FUNCTION_BLOCK FB_Conveyor
VAR CONSTANT
	sCycleStateTextDef: ARRAY[0..10]  OF STRING :=	
		['State 0: Wait for Start',
		'State 1: Start conveyor',
		'State 2: Start Gantries',
		'State 3: Spare',
		'State 4: Spare',
		'State 5: Spare',
		'State 6: Belt running, control speed','7','8','9',
		'State 10: Error'];
	
	tCycleStateTimeouts: ARRAY[0..10] OF TIME := 
		[T#10S,T#10S,T#60S,T#10S,T#10S,T#10S,T#10S,T#10S,T#10S,T#10S,
		T#10S];

END_VAR
VAR_INPUT
	mxResetCycleState				: BOOL;
	mxReset							: BOOL;	(*Reset Error*)
	mxEmergency						: BOOL;
	mxAutoMode						: BOOL; (* TRUE = Automode *)
	mxFirstCycle					: BOOL;

END_VAR
VAR_IN_OUT
	MachParameters					: ST_ConveyorMachPar;
	ProdParameters					: ST_ConveyorProdPar;
	SysParameters					: ST_ConveyorSysPar;
	
	IMD1_COM_IN						: ST_COM_IMD_SpdCntrl;
	IMD1_COM_OUT					: ST_COM_SpdCntrl_IMD;
	IMD2_COM_IN						: ST_COM_IMD_SpdCntrl;
	IMD2_COM_OUT					: ST_COM_SpdCntrl_IMD;
	
	FTL_COM_IN						: ST_COM_FTL_SpdCntrl;
	FTL_COM_OUT						: ST_COM_SpdCntrl_FTL;
END_VAR
VAR_OUTPUT
	(*Errors*)
	Errors							: ST_ConveyorErrors;
	mxErrorInit						: BOOL;
	mxErrorStopinPos				: BOOL;		(* Error, stop in position. Only reset neccesary *)

(* State vars *)
	mxCycleBusy						: BOOL;
	
(* Vars *)	
	mrActModPos						: LREAL;
END_VAR
VAR
(* State vars *)
	miCycleState					: INT :=0;
	miCycleOldstate					: INT :=0;
	mxCycleTransitionState			: BOOL := FALSE;
	sCycleStateText					: STRING;
	exCycleTimeOut					: BOOL;		(* Timeout for the whole programcycle *)
	CycleTimeout					: TON;
	CycleTimeOutUpFlank				: R_TRIG;
	mxCycleTimeoutEnable			: BOOL;
	CycleTime						: REAL;
	mxCycleHasError					: BOOL;
	miStopState						: INT;
	mxStartCycle					: BOOL;
	mxStopCycle						: BOOL;
	mxStopDirect					: BOOL;
	
	(* Objects *)
	Belt							: FB_NcAxis;
	IMD1_GantryA					: FB_BlowOff;
	IMD1_GantryB					: FB_BlowOff;
	IMD2_GantryA					: FB_BlowOff;
	IMD2_GantryB					: FB_BlowOff;

	mrSetpointPosition				: LREAL;
	mrActPosBeltSaved				: LREAL;	
	
	(* Internal calculating values *)
	mrModuloStart_offset			: LREAL;
	mdModuloCount					: DINT;
	RT_ModuloCount					: R_TRIG;
	mrCalculateSpeedIMD1			: LREAL;
	mrCalculateSpeedIMD2			: LREAL;
	mrAllowdKObyFTL					: LREAL;
	mrCalculateSpeedFTL				: LREAL;
	StartSpeedConveyorAuto			: LREAL;	
	mrSetRunSpeed					: LREAL;	
	miNrOfIMD						: INT := 2; //Always calculate based on two IMD enabled
	mrSetRunSpeedOld				: LREAL;
	T_Stopping						: TON;
END_VAR

mrActModPos:= Belt.axAxis.NcToPlc.ModuloActPos;

Error();
Cycle();
Objects();

ACTION Cycle:
(*StateChange (Transition)  Signalgeneration*)
mxCycleTransitionState:=(miCycleState<>miCycleOldstate);
(*State text*)
sCycleStateText:=sCycleStateTextDef[miCycleState];
(*Timeout Watchdog for Statemachine*)
mxCycleTimeoutEnable:=NOT (miCycleState=0 OR miCycleState=6) AND NOT mxReset;

CycleTimeout(IN:=mxCycleTimeoutEnable, PT:=tCycleStateTimeouts[miCycleState] );
CycleTimeOutUpFlank(CLK:=CycleTimeout.Q );
miCycleOldstate:=miCycleState;

(*Set Errorbit when Raising edge of Timeout has been detected*)
IF CycleTimeOutUpFlank.Q THEN
	exCycleTimeOut:=TRUE; 			(* 1 Timeout for the whole programcycle *)
END_IF

(*Function to reset the Statemachine*)
IF mxResetCycleState THEN
	mxResetCycleState:= FALSE;
	miCycleState:=0;
	miCycleOldstate:=miCycleState;
	mxCycleTransitionState:=FALSE;
	mdModuloCount := 0;
	
	IMD1_GantryA.mxResetCycleState := TRUE;
	IMD1_GantryB.mxResetCycleState := TRUE;
	IMD2_GantryA.mxResetCycleState := TRUE;
	IMD2_GantryB.mxResetCycleState := TRUE;
	
	T_Stopping.IN := FALSE;
	IMD1_COM_OUT.StopForming := FALSE;
    IMD2_COM_OUT.StopForming := FALSE;
		
	mxStartCycle:= FALSE;
	mxStopCycle:= FALSE;
	mxStopDirect:= FALSE;
	Belt.M_Stop();
END_IF

(*Definition State has Error*)
mxCycleHasError:=FALSE;

(*Calculate modulo offset positions gantry*)
	IF ProdParameters.BlowOff_Prod.Modulo = 0 THEN
		ProdParameters.BlowOff_Prod.Modulo := 4620;
	END_IF
	IMD1_GantryA.mrModuloOffset:= (ProdParameters.BlowOff_Prod.Modulo/4)*1;
	IMD1_GantryB.mrModuloOffset:= (ProdParameters.BlowOff_Prod.Modulo/4)*3;
	IMD2_GantryA.mrModuloOffset:= 0;
	IMD2_GantryB.mrModuloOffset:= (ProdParameters.BlowOff_Prod.Modulo/4)*2;

(*Calculate allowed speeds from Communication partners *)
	(*IF MachParameters.IMD1_Enabled AND MachParameters.IMD2_Enabled THEN		//For now speed of the conveyor will always be based on 2 IMD's
		miNrOfIMD := 2;
	ELSIF MachParameters.IMD1_Enabled OR MachParameters.IMD2_Enabled THEN
		miNrOfIMD := 1;	
	END_IF*)
	
	IF ProdParameters.BlowOff_Prod.NrOfSheets = 0 THEN
		ProdParameters.BlowOff_Prod.NrOfSheets := 3;
	END_IF
	
	IF ((IMD1_COM_IN.MaximumSpeed = 0) AND IMD1_COM_IN.RTO) THEN
		mrCalculateSpeedIMD1 := StartSpeedConveyorAuto;
	ELSE
		mrCalculateSpeedIMD1 := ((IMD1_COM_IN.MaximumSpeed-0.05) * miNrOfIMD)*((ProdParameters.BlowOff_Prod.Modulo/4)/60);
	END_IF
	IF ((IMD2_COM_IN.MaximumSpeed = 0) AND IMD2_COM_IN.RTO) THEN
		mrCalculateSpeedIMD2 := StartSpeedConveyorAuto;
	ELSE
		mrCalculateSpeedIMD2 := ((IMD2_COM_IN.MaximumSpeed-0.05) * miNrOfIMD)*((ProdParameters.BlowOff_Prod.Modulo/4)/60);	
	END_IF
	mrAllowdKObyFTL := (FTL_COM_IN.MaximumSpeed/ProdParameters.BlowOff_Prod.NrOfSheets)/miNrOfIMD; 	
	mrCalculateSpeedFTL := (mrAllowdKObyFTL * miNrOfIMD)*((ProdParameters.BlowOff_Prod.Modulo/4)/60);
	StartSpeedConveyorAuto := (MachParameters.VelocityAuto * miNrOfIMD)*((ProdParameters.BlowOff_Prod.Modulo/4)/60);
	IF StartSpeedConveyorAuto > mrCalculateSpeedFTL THEN
		StartSpeedConveyorAuto := mrCalculateSpeedFTL;
	END_IF
	
	IF (MachParameters.IMD1_Enabled AND IMD1_COM_IN.RTO) AND (MachParameters.IMD2_Enabled AND IMD2_COM_IN.RTO) THEN
		IF ( mrCalculateSpeedIMD1 <= mrCalculateSpeedFTL ) AND (mrCalculateSpeedIMD2 <= mrCalculateSpeedFTL) THEN
			IF (mrCalculateSpeedIMD1 <= mrCalculateSpeedIMD2) THEN
				mrSetRunSpeed := mrCalculateSpeedIMD1;
			ELSE
				mrSetRunSpeed := mrCalculateSpeedIMD2;
			END_IF
		ELSIF ( mrCalculateSpeedIMD1 <= mrCalculateSpeedFTL ) AND (mrCalculateSpeedIMD2 >= mrCalculateSpeedFTL) THEN
			mrSetRunSpeed := mrCalculateSpeedIMD1;
		ELSIF ( mrCalculateSpeedIMD1 >= mrCalculateSpeedFTL ) AND (mrCalculateSpeedIMD2 <= mrCalculateSpeedFTL) THEN
			mrSetRunSpeed := mrCalculateSpeedIMD2;
		ELSE
			mrSetRunSpeed := mrCalculateSpeedFTL;
		END_IF	
	ELSIF MachParameters.IMD1_Enabled AND IMD1_COM_IN.RTO THEN
		IF mrCalculateSpeedIMD1 <= mrCalculateSpeedFTL THEN
			mrSetRunSpeed := mrCalculateSpeedIMD1;
		ELSE
			mrSetRunSpeed := mrCalculateSpeedFTL;
		END_IF
	ELSIF MachParameters.IMD2_Enabled AND IMD2_COM_IN.RTO THEN
		IF mrCalculateSpeedIMD2 <= mrCalculateSpeedFTL THEN
			mrSetRunSpeed := mrCalculateSpeedIMD2;
		ELSE
			mrSetRunSpeed := mrCalculateSpeedFTL;
		END_IF
	ELSIF NOT IMD1_COM_IN.RTO AND NOT IMD2_COM_IN.RTO THEN
		mrSetRunSpeed := StartSpeedConveyorAuto;	
	END_IF
	IF mrSetRunSpeed < StartSpeedConveyorAuto AND (( MachParameters.IMD1_Enabled AND IMD1_COM_IN.RTO) OR (MachParameters.IMD2_Enabled AND IMD2_COM_IN.RTO)) THEN
			mrSetRunSpeed := StartSpeedConveyorAuto;
	END_IF
	
(*Time delay speed control stopped to IMD's*)
	T_Stopping(PT:=T#5S);
	IF T_Stopping.Q THEN
		IMD1_COM_OUT.StopForming := TRUE;
        IMD2_COM_OUT.StopForming := TRUE;
	END_IF
	
(*Cycle State's*)
CASE miCycleState OF
	0:
	(*
		- wait for startcycle
		- Move belt with velo
  
	*)
		IF mxStartCycle THEN
			mxStartCycle:= FALSE;
			T_Stopping.IN := FALSE;
			IMD1_COM_OUT.StopForming := FALSE;
            IMD2_COM_OUT.StopForming := FALSE;
			
			miCycleState:= 1;
		END_IF	

	(* Move belt *)
	1:
		IF mxStopDirect THEN
			mxStopDirect:= FALSE;
			
			miCycleState:= 25;
		ELSIF mxStopCycle THEN
			mxStopCycle:= FALSE;

			mrActPosBeltSaved:= Belt.ActPosition;		
	
			miStopState:= miCycleState;
			miCycleState:= 20;
		ELSIF FTL_COM_IN.RTO THEN
			mdModuloCount := 0;
			IF StartSpeedConveyorAuto > mrCalculateSpeedFTL THEN
				mrSetRunSpeed := mrCalculateSpeedFTL;
			ELSE
				mrSetRunSpeed := StartSpeedConveyorAuto;
			END_IF
			Belt.M_MoveVelocity(Velocity:= mrSetRunSpeed, Direction:= MC_Positive_Direction);
	
			miCycleState := 2;
				
		END_IF
		
	(* Start first Gantry *)	
	2:	
		IF mxStopDirect THEN
			mxStopDirect:= FALSE;
			
			miCycleState:= 25;
		ELSIF mxStopCycle THEN
			mxStopCycle:= FALSE;

			mrActPosBeltSaved:= Belt.ActPosition;		
	
			miStopState:= miCycleState;
			miCycleState:= 20;
		ELSE
		
			IF mrActModPos >= (IMD2_GantryA.mrModuloOffset - mrModuloStart_offset) AND  mrActModPos <= (IMD2_GantryA.mrModuloOffset + mrModuloStart_offset) THEN
				IMD2_GantryA.M_StartCycle();
			ELSIF mrActModPos >= (IMD1_GantryA.mrModuloOffset - mrModuloStart_offset) AND  mrActModPos <= (IMD1_GantryA.mrModuloOffset + mrModuloStart_offset) THEN
				IMD1_GantryA.M_StartCycle();
			ELSIF mrActModPos >= (IMD2_GantryB.mrModuloOffset - mrModuloStart_offset) AND  mrActModPos <= (IMD2_GantryB.mrModuloOffset + mrModuloStart_offset) THEN
				IMD2_GantryB.M_StartCycle();		
			ELSIF mrActModPos >= (IMD1_GantryB.mrModuloOffset - mrModuloStart_offset) AND  mrActModPos <= (IMD1_GantryB.mrModuloOffset + mrModuloStart_offset) THEN
				IMD1_GantryB.M_StartCycle();			
			END_IF
			
			IF IMD1_GantryA.mxCycleBusy AND IMD1_GantryB.mxCycleBusy AND IMD2_GantryA.mxCycleBusy AND IMD2_GantryB.mxCycleBusy THEN
				miCycleState:= 6;
			END_IF

		END_IF
	
		
	(* Speed control *)	
	6:
		IF mxStopDirect THEN
			mxStopDirect:= FALSE;
			
			miCycleState:= 25;
		ELSIF mxStopCycle THEN
			mxStopCycle:= FALSE;

			mrActPosBeltSaved:= Belt.ActPosition;		
	
			miStopState:= miCycleState;
			miCycleState:= 20;
		ELSE
			RT_ModuloCount(CLK:= mrActModPos >= (ProdParameters.BlowOff_Prod.Modulo - ProdParameters.BlowOff_Prod.PitchGantry));
			IF 	RT_ModuloCount.Q THEN
				mdModuloCount := mdModuloCount + 1;
			END_IF
			(*IF (Belt.ActVelocity < mrSetRunSpeed) AND (mrSetRunSpeed > 0) THEN
				Belt.M_MoveVelocity(Velocity:= mrSetRunSpeed, Direction:= MC_Positive_Direction);
			END_IF*)
			IF (mdModuloCount >=  MachParameters.ModuloRamp) OR (mrSetRunSpeed = mrCalculateSpeedFTL) OR (mrSetRunSpeed < mrSetRunSpeedOld) THEN
				mdModuloCount := 0;
				Belt.M_MoveVelocity(Velocity:= mrSetRunSpeed, Direction:= MC_Positive_Direction);
			END_IF			
		END_IF	
		
	
	(* Stop Cycle, stop belt after x mm*)
	20:
		IF mxStopDirect THEN
			mxStopDirect:= FALSE;
			
			miCycleState:= 25;
		ELSE 
			mxStopCycle:= FALSE;
			mdModuloCount := 0;
			
			Belt.M_Stop();	
			IMD1_GantryA.M_StopCycle();
			IMD1_GantryB.M_StopCycle();
			IMD2_GantryA.M_StopCycle();
			IMD2_GantryB.M_StopCycle();
			T_Stopping.IN := TRUE;
			//IMD1_COM_OUT.StopForming := TRUE;
			//IMD2_COM_OUT.StopForming := TRUE;
			
			IF NOT Belt.axStatus.Moving OR Belt.axStatus.StandStill THEN		
				miCycleState:= 21;
			END_IF
		END_IF

	21:
		IF mxStopDirect THEN
			mxStopDirect:= FALSE;
			
			miCycleState:= 25;
		ELSIF mxStartCycle THEN		
			T_Stopping.IN := FALSE;	
			mxStartCycle := FALSE;
			
			miCycleState:= 22;			
		END_IF
	
	(* wait for FTL *)	
	22:
		IF mxStopDirect THEN
			mxStopDirect:= FALSE;
			
			miCycleState:= 25;
		ELSIF FTL_COM_IN.RTO THEN		

			IMD1_GantryA.M_StartCycle();
			IMD1_GantryB.M_StartCycle();
			IMD2_GantryA.M_StartCycle();
			IMD2_GantryB.M_StartCycle();
			
			IMD1_COM_OUT.StopForming := FALSE;
			IMD2_COM_OUT.StopForming := FALSE;
			
			IF StartSpeedConveyorAuto > mrCalculateSpeedFTL THEN
				mrSetRunSpeed := mrCalculateSpeedFTL;
			ELSE
				mrSetRunSpeed := StartSpeedConveyorAuto;
			END_IF
			Belt.M_MoveVelocity(Velocity:= mrSetRunSpeed, Direction:= MC_Positive_Direction);
			
			miCycleState:= miStopState;			
		END_IF

	(* Stop Direct *)
	25:			
		mxStartCycle:= FALSE;
		mxStopCycle:= FALSE;
		mxStopDirect:= FALSE;
		mdModuloCount := 0;
		
		IMD1_GantryA.M_StopDirect();
		IMD1_GantryB.M_StopDirect();
		IMD2_GantryA.M_StopDirect();
		IMD2_GantryB.M_StopDirect();
		
		T_Stopping.IN := TRUE;
		//IMD1_COM_OUT.StopForming := TRUE;
		//IMD2_COM_OUT.StopForming := TRUE;
		
		Belt.M_Stop();

		miCycleState:= 0;
END_CASE

mxCycleBusy:= miCycleState<>0 AND miCycleState <>21;
IMD1_COM_OUT.Modulo := IMD2_COM_OUT.Modulo := mrActModPos;
IMD1_COM_OUT.SpeedInKo := IMD2_COM_OUT.SpeedInKo := (mrSetRunSpeed/((ProdParameters.BlowOff_Prod.Modulo/4)/60))/miNrOfIMD;
mrSetRunSpeedOld := mrSetRunSpeed;
END_ACTION

ACTION Error:


(*************************************************************************************************)
mxErrorStopinPos:= Belt.ErrorStop;
END_ACTION

METHOD M_StartCycle

IF NOT mxCycleBusy THEN
	mxStartCycle:= TRUE;	
END_IF
END_METHOD

METHOD M_StopCycle

IF mxCycleBusy THEN 
	mxStopCycle:= TRUE; 
END_IF
END_METHOD

METHOD M_StopDirect

IF mxCycleBusy THEN
	mxStopDirect:= TRUE;	
END_IF
END_METHOD

ACTION Objects:
IMD1_GantryA(
	mxReset							:= mxReset,
	mxEmergency						:= mxEmergency,
	mxAutoMode						:= mxAutoMode,
	mrActModulo						:= mrActModPos,
	ProdPar							:= ProdParameters.BlowOff_Prod,
	COM_IMD_Stopped					:= IMD1_COM_IN.Stopped,
	COM_IMD_RTO						:= IMD1_COM_IN.RTO,
	COM_StartFormingReady			:= IMD1_COM_IN.FormingReadyA,
	COM_BlownOffProcessed			:= IMD1_COM_IN.BlowOffProcessedA,
	COM_GantryInPos 				:= IMD1_COM_IN.GantryA_Ready,
	COM_BlowOff_Pulse				=> IMD1_COM_OUT.BlowOffPulseA,
	COM_StartForming				=> IMD1_COM_OUT.StartFormingA, 
	COM_ErrSlotNotFree				=> IMD1_COM_OUT.ErrSlotANotFree,
);                                  

IMD1_GantryB(
	mxReset							:= mxReset,
	mxEmergency						:= mxEmergency,
	mxAutoMode						:= mxAutoMode,
	mrActModulo						:= mrActModPos,
	ProdPar							:= ProdParameters.BlowOff_Prod,
	COM_IMD_Stopped					:= IMD1_COM_IN.Stopped,
	COM_IMD_RTO						:= IMD1_COM_IN.RTO,
	COM_StartFormingReady			:= IMD1_COM_IN.FormingReadyB,
	COM_BlownOffProcessed			:= IMD1_COM_IN.BlowOffProcessedB,
	COM_GantryInPos 				:= IMD1_COM_IN.GantryB_Ready,
	COM_BlowOff_Pulse				=> IMD1_COM_OUT.BlowOffPulseB,
	COM_StartForming				=> IMD1_COM_OUT.StartFormingB, 
	COM_ErrSlotNotFree				=> IMD1_COM_OUT.ErrSlotBNotFree
); 


IMD2_GantryA(
	mxReset							:= mxReset,
	mxEmergency						:= mxEmergency,
	mxAutoMode						:= mxAutoMode,
	mrActModulo						:= mrActModPos,
	ProdPar							:= ProdParameters.BlowOff_Prod,
	COM_IMD_Stopped					:= IMD2_COM_IN.Stopped,
	COM_IMD_RTO						:= IMD2_COM_IN.RTO,
	COM_StartFormingReady			:= IMD2_COM_IN.FormingReadyA,
	COM_BlownOffProcessed			:= IMD2_COM_IN.BlowOffProcessedA,
	COM_GantryInPos 				:= IMD2_COM_IN.GantryA_Ready,
	COM_BlowOff_Pulse				=> IMD2_COM_OUT.BlowOffPulseA,
	COM_StartForming				=> IMD2_COM_OUT.StartFormingA, 
	COM_ErrSlotNotFree				=> IMD2_COM_OUT.ErrSlotANotFree
); 

IMD2_GantryB(
	mxReset							:= mxReset,
	mxEmergency						:= mxEmergency,
	mxAutoMode						:= mxAutoMode,
	mrActModulo						:= mrActModPos,
	ProdPar							:= ProdParameters.BlowOff_Prod,
	COM_IMD_Stopped					:= IMD2_COM_IN.Stopped,
	COM_IMD_RTO						:= IMD2_COM_IN.RTO,
	COM_StartFormingReady			:= IMD2_COM_IN.FormingReadyB,
	COM_BlownOffProcessed			:= IMD2_COM_IN.BlowOffProcessedB,
	COM_GantryInPos 				:= IMD2_COM_IN.GantryB_Ready,
	COM_BlowOff_Pulse				=> IMD2_COM_OUT.BlowOffPulseB,
	COM_StartForming				=> IMD2_COM_OUT.StartFormingB, 
	COM_ErrSlotNotFree				=> IMD2_COM_OUT.ErrSlotBNotFree
); 

Belt(
	mxEnable:= NOT mxEmergency, 
	mxInhibit:= FALSE, 
	mxAutoMode:= mxAutoMode, 
	mxReset:= mxReset, 
	mxEmergency:= mxEmergency, 
	mxSimulation:= , 
	mxFirstCycle:= , 
	mxResetCycle:= , 
	mxDisable_Positive:= FALSE, 
	mxDisable_Negative:= FALSE, 
	mxBlockHMI:= , 
	mrOverride:= 100.0, 
	mrVelocityManual:= MachParameters.VelocityManual, 
	SysParameters:= SysParameters.Belt,
	mxCycleBusy=> , 
	mxRunning=> , 
	Errors=> Errors.NCAxisError, 
	Error=> , 
	ErrorStop=> , 
	axStatus=> , 
	ActPosition=> , 
	ActVelocity=> , 
	axAxis=> );
END_ACTION

END_FUNCTION_BLOCK

(* stored: Version 1.1.0.1, ProductVersion 3.1.4020.12
   POU FB_Conveyor: Id {2f00a41b-0680-4725-a9db-8bcc4a3809de}, SpecialFunc None
   Action Cycle: Id {e859f666-04a5-47c3-aeb6-4a0a8e295096}
   Action Error: Id {4acfcdbf-3042-407f-b5fd-c5a660e19f95}
   Method M_StartCycle: Id {31ade575-aaa5-48b4-9916-2fbf369914dc}
   Method M_StopCycle: Id {1a479aea-c5e5-4972-955a-2ca3d3ef1ab4}
   Method M_StopDirect: Id {b6cb47ae-764b-4727-b4c1-ac0c79561633}
   Action Objects: Id {c720eaca-4841-47e7-b3ea-ce50545180c4} *)
